// This function has been automatically generated from the project information.
{attribute 'signature_flag' := '1073741824'}
{attribute 'TcGenerated'}
{attribute 'no-analysis'}
FUNCTION F_GetVersion : ST_LibVersion
VAR_INPUT
	
END_VAR

F_GetVersion.iMajor := 0;
F_GetVersion.iMinor := 2;
F_GetVersion.iBuild := 0;
F_GetVersion.iRevision := 1;

END_FUNCTION

(* stored: Version 1.1.0.1
   POU F_GetVersion: Id {e2f318b7-74dd-0bf5-2305-50e9fb98b9ad}, SpecialFunc None *)
